// Mitsubishi GX Works2 project: PID   PLC: FX3G
// Базовая структура управления вентиляциооной установкой

// global labels: Global1
VAR_GLOBAL
  PID_PV AT R110 : INT;
  TempSupply AT R100 : INT;
  xMode AT M500 : BOOL;
  xStart AT M501 : BOOL;
  xAT AT M502 : BOOL;
  xATMode AT M503 : BOOL;
  iDelta AT R102 : INT;
  Setpoint AT R101 : INT;
  TempOut AT R103 : INT;
  Kp AT D150 : INT;
  Ti AT D151 : INT;
  Kd AT D152 : INT;
  Td AT D153 : INT;
  xInit AT M504 : BOOL;
  Timer_1 AT K100 : INT;
  Timer_out AT K105 : INT;
  myTON : myTON;
  progTON : TON;
  myTON_Q AT M498 : BOOL;
  progTON_Q AT M499 : BOOL;
END_VAR

// task Task_01 (event TRUE, interval 0, priority 31): POU_01
// task Init (event M8002, interval 0, priority 24): 
// task Process (event FALSE, interval T#150ms, priority 29): 
// user libraries (not included): Timers

PROGRAM POU_01
VAR
  R_TRIG_1 : R_TRIG;
END_VAR
(* TP(IN:= xStart ,PT:= T#2sec ,Q:= xInit ); *)
IF xStart THEN 
		R500 := 2#0000000000000001;
		R501 := 2#0000000001110001;
		R502 := 30;
		R522 := 100;
		R523 := 0;
		R525 := iDelta;
		R526 := 100;
		R527 := 0;
END_IF; 


progTON(IN:= xStart ,PT:=T#12s ,Q:= progTON_Q );
IF MEF(xStart) THEN progTON(IN:= FALSE ,PT:=T#0ms ,Q:= progTON_Q ); END_IF; 

		PID( xStart , Setpoint , TempSupply , R500 , PID_PV );
END_PROGRAM

FUNCTION SeasonControl
VAR_INPUT
  tempOut : INT;  (* Temp Outdore - Температура наружнего воздуха *)
  tempWinter : INT;  (* Temp for switch on Winter - Уставка перехода на Зимний режим *)
  tempSummer : INT;  (* Temp for switch on Summer - Уставка перехода на летний режим *)
  triger : BOOL;  (* 1 - was switch to winter 0 - was switch to summer *)
END_VAR
IF tempOut  <  tempWinter THEN 
		SeasonControl := 1; (* Output  Set flag - 1  to force switching to Winter *)
	ELSE 
		IF tempOut  > tempSummer THEN 
			SeasonControl := 0; (* Output  Set flag - 0  to force switching to Summer*)
		ELSE 
			SeasonControl := triger; (* Don't change r*)
		END_IF;

	END_IF;
END_FUNCTION

FUNCTION TestFunction
TestFunction := TRUE;
END_FUNCTION
